// TIA Portal project "SCL EJERCICIO 4" (V11)

(* hardware
DEVICE "S7300/ET200 station_1"  SIMATIC 300-Station
   slot 0: "Perfil soporte_0"  Rail  6ES7 390-1***0-0AA0
   slot 2: "PLC_1"  CPU 313C-2 DP  6ES7 313-6CF03-0AB0  V2.6
      slot 0: "Interfaz MPI_1"  MPI
      slot 1: "Interfaz DP_1"  DP
      slot 2: "DI16/DO16_1"  DI16/DO16
      slot 4: "Contaje_1"  Counter
*)

// ===== PLC "PLC_1"  CPU 313C-2 DP =====

VAR_GLOBAL   // PLC tag table "Tabla de variables estándar"
   "Tag_1" AT %A0.0 : Bool;
   "Tag_2" AT %A0.1 : Bool;
   "Tag_3" AT %A0.2 : Bool;
   "Tag_4" AT %A0.3 : Bool;
   "Tag_5" AT %A0.4 : Bool;
   "Tag_6" AT %A0.5 : Bool;
   "Tag_7" AT %E0.0 : Bool;
   "Tag_8" AT %T0 : Timer;
   "Tag_9" AT %T2 : Timer;
   "Tag_10" AT %T3 : Timer;
   "Tag_11" AT %T4 : Timer;
END_VAR

DATA_BLOCK "SEMAFORO_DB_2"   // DB3
{ S7_Optimized_Access := 'FALSE' }
VERSION : 0.1
// stored: InstanceOfName SEMAFORO
"SEMAFORO"
BEGIN
END_DATA_BLOCK

FUNCTION_BLOCK "SEMAFORO"   // FB1, SCL
{ S7_Optimized_Access := 'FALSE' }
VERSION : 0.1
   VAR_OUTPUT
      "s1 verde" : Bool;
      "s1 ambar" : Bool;
      "s1 rojo" : Bool;
      "s2 verde" : Bool;
      "s2 ambar" : Bool;
      "s2 rojo" : Bool;
   END_VAR
   VAR
      M0 : Bool;
      M1 : Bool;
      t0 : Bool;
      "VISUALIZAR 0" : Time;
      t1 : Bool;
      "VISUALIZAR 1" : Time;
      t2 : Bool;
      "VISUALIZAR 2" : Time;
      t3 : Bool;
      "VISUALIZAR 3" : Time;
      t4 : Bool;
      "VISUALIZAR 4" : Time;
      t5 : Bool;
      "VISUALIZAR 5" : Time;
   END_VAR
BEGIN
   IF NOT #M0   THEN (* encendido incial sin actuar con ningun pulsador *)
     #"s1 verde":=true;
     #"s2 rojo":=true;
     #M0:=TRUE;
   END_IF;
   "IEC_Timer_0_DB".TON(IN:=#"s1 verde",(*temporizado cambio color 1 *)
                        PT:=t#20s,
                        Q=>#t0,
                        ET=>#"VISUALIZAR 0");

   IF #t0 THEN (* semaforo 1 cambio verde a ambar *)
      #"s1 verde":=false;
     #"s1 ambar":=true;
     END_IF;

   "IEC_Timer_0_DB_1".TON(IN:=#"s1 ambar",(* temporizado cambio de color 2*)
                          PT:=T#3S,
                          Q=>#t1,
                          ET=>#"VISUALIZAR 1");

   IF #t1 THEN (* semaforo 1 cambio ambar a rojo *)
     #"s1 ambar":=false;
     #"s1 rojo":=true;
   END_IF;

   "IEC_Timer_0_DB_3".TON(IN:=#"s1 rojo",(* temporizado cambio de color 3 *)
                          PT:=T#2S,
                          Q=>#t2,
                          ET=>#"VISUALIZAR 2");

   IF #t2 THEN (* semaforo 2 cambio rojo a verde *)
     #"s2 rojo":=false;
     #"s2 verde" :=true;
   END_IF;

   "IEC_Timer_0_DB_2".TON(IN:= #"s2 verde",(* temporizado cambio de color 4 *)
                          PT:=T#18S,
                          Q=>#t3,
                          ET=>#"VISUALIZAR 3");

   IF #t3 THEN (* semaforo 2 cambio verde a ambar *)
       #"s2 verde":=false;
     #"s2 ambar":=true;
   END_IF;

   "IEC_Timer_0_DB_4".TON(IN:=#"s2 ambar", (* temporizado cambio de color 5 *)
                          PT:=t#3s,
                          Q=>#t4,
                          ET=>#"VISUALIZAR 4");

   IF #t4 THEN (* semaforo 2 cambio de ambar a rojo*)
     #"s2 ambar":=false;
     #"s2 rojo" :=true;
     #M1:=TRUE;
      END_IF;

   "IEC_Timer_0_DB_5".TON(IN:= #M1, (*temporizdo cambio de color 6 *)
                          PT:=T#2S,
                          Q=>#t5,
                          ET=>#"VISUALIZAR 5");

   IF #t5 THEN (*reinicio de ciclo permanene *) 
     #M1:=FALSE;
     #"s1 rojo":=FALSE;
     #"s1 verde":=TRUE;
   END_IF;
END_FUNCTION_BLOCK

ORGANIZATION_BLOCK "Main"   // OB1, LAD
TITLE = "Main Program Sweep (Cycle)"
{ S7_Optimized_Access := 'FALSE' }
VERSION : 0.1
   VAR_TEMP
      OB1_EV_CLASS : Byte;   // Bits 0-3 = 1 (Coming event), Bits 4-7 = 1 (Event class 1)
      OB1_SCAN_1 : Byte;   // 1 (Cold restart scan 1 of OB 1), 3 (Scan 2-n of OB 1)
      OB1_PRIORITY : Byte;   // Priority of OB Execution
      OB1_OB_NUMBR : Byte;   // 1 (Organization block 1, OB1)
      OB1_RESERVED_1 : Byte;   // Reserved for system
      OB1_RESERVED_2 : Byte;   // Reserved for system
      OB1_PREV_CYCLE : Int;   // Cycle time of previous OB1 scan (milliseconds)
      OB1_MIN_CYCLE : Int;   // Minimum cycle time of OB1 (milliseconds)
      OB1_MAX_CYCLE : Int;   // Maximum cycle time of OB1 (milliseconds)
      OB1_DATE_TIME : Date_And_Time;   // Date and time OB1 started
   END_VAR
BEGIN

REGION Network 1
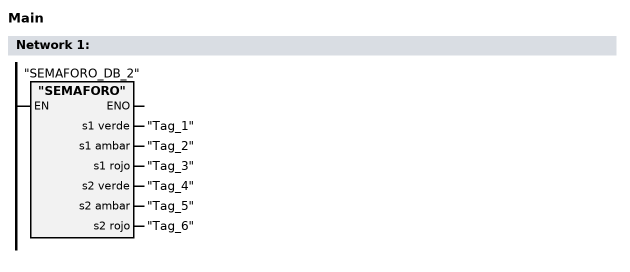
   RUNG wire#powerrail
      "SEMAFORO_DB_2"("s1 verde" => "Tag_1", "s1 ambar" => "Tag_2", "s1 rojo" => "Tag_3", "s2 verde" => "Tag_4", "s2 ambar" => "Tag_5", "s2 rojo" => "Tag_6")
   END_RUNG
   // the same network as SCL:
   "SEMAFORO_DB_2"("s1 verde" => "Tag_1",   // "SEMAFORO"
                   "s1 ambar" => "Tag_2",
                   "s1 rojo" => "Tag_3",
                   "s2 verde" => "Tag_4",
                   "s2 ambar" => "Tag_5",
                   "s2 rojo" => "Tag_6");
END_REGION
END_ORGANIZATION_BLOCK